// TIA Portal project "Project2" (V20)

(* hardware
DEVICE "S7-300/ET200M station_1"  S7-300 station
   slot 0: "Rail_0"  Rail  6ES7 390-1***0-0AA0
   slot 2: "PLC_1"  CPU 312  6ES7 312-1AE14-0AB0  V3.3
      slot 0: "MPI interface_1"  MPI
*)

// ===== PLC "PLC_1"  CPU 312 =====

ORGANIZATION_BLOCK "Main"   // OB1, LAD
TITLE = "Main Program Sweep (Cycle)"
{ S7_Optimized_Access := 'FALSE' }
VERSION : 0.1
   VAR_TEMP
      OB1_EV_CLASS : Byte;   // Bits 0-3 = 1 (Coming event), Bits 4-7 = 1 (Event class 1)
      OB1_SCAN_1 : Byte;   // 1 (Cold restart scan 1 of OB 1), 3 (Scan 2-n of OB 1)
      OB1_PRIORITY : Byte;   // Priority of OB Execution
      OB1_OB_NUMBR : Byte;   // 1 (Organization block 1, OB1)
      OB1_RESERVED_1 : Byte;   // Reserved for system
      OB1_RESERVED_2 : Byte;   // Reserved for system
      OB1_PREV_CYCLE : Int;   // Cycle time of previous OB1 scan (milliseconds)
      OB1_MIN_CYCLE : Int;   // Minimum cycle time of OB1 (milliseconds)
      OB1_MAX_CYCLE : Int;   // Maximum cycle time of OB1 (milliseconds)
      OB1_DATE_TIME : Date_And_Time;   // Date and time OB1 started
      S6 : Bool;
      S7 : Bool;
      S8 : Bool;
      "S1(sus stanga)" : Bool;
      "S2(sus Dreapta)" : Bool;
      "S3(jos stanga)" : Bool;
      "S4(jos Dreapta)" : Bool;
      "S5(soft reset)" : Bool;
      "S0(Hard reset)" : Bool;
      eroare : Bool;
      P1 : Bool;
      P2 : Bool;
      P3 : Bool;
      P4 : Bool;
      alarma : Bool;
   END_VAR
   VAR_TEMP   // added for the SCL form of the ladder/FBD networks
      _w1 : Bool;
      _w2 : Bool;
      _w3 : Bool;
      _w4 : Bool;
   END_VAR
BEGIN

REGION Network 1
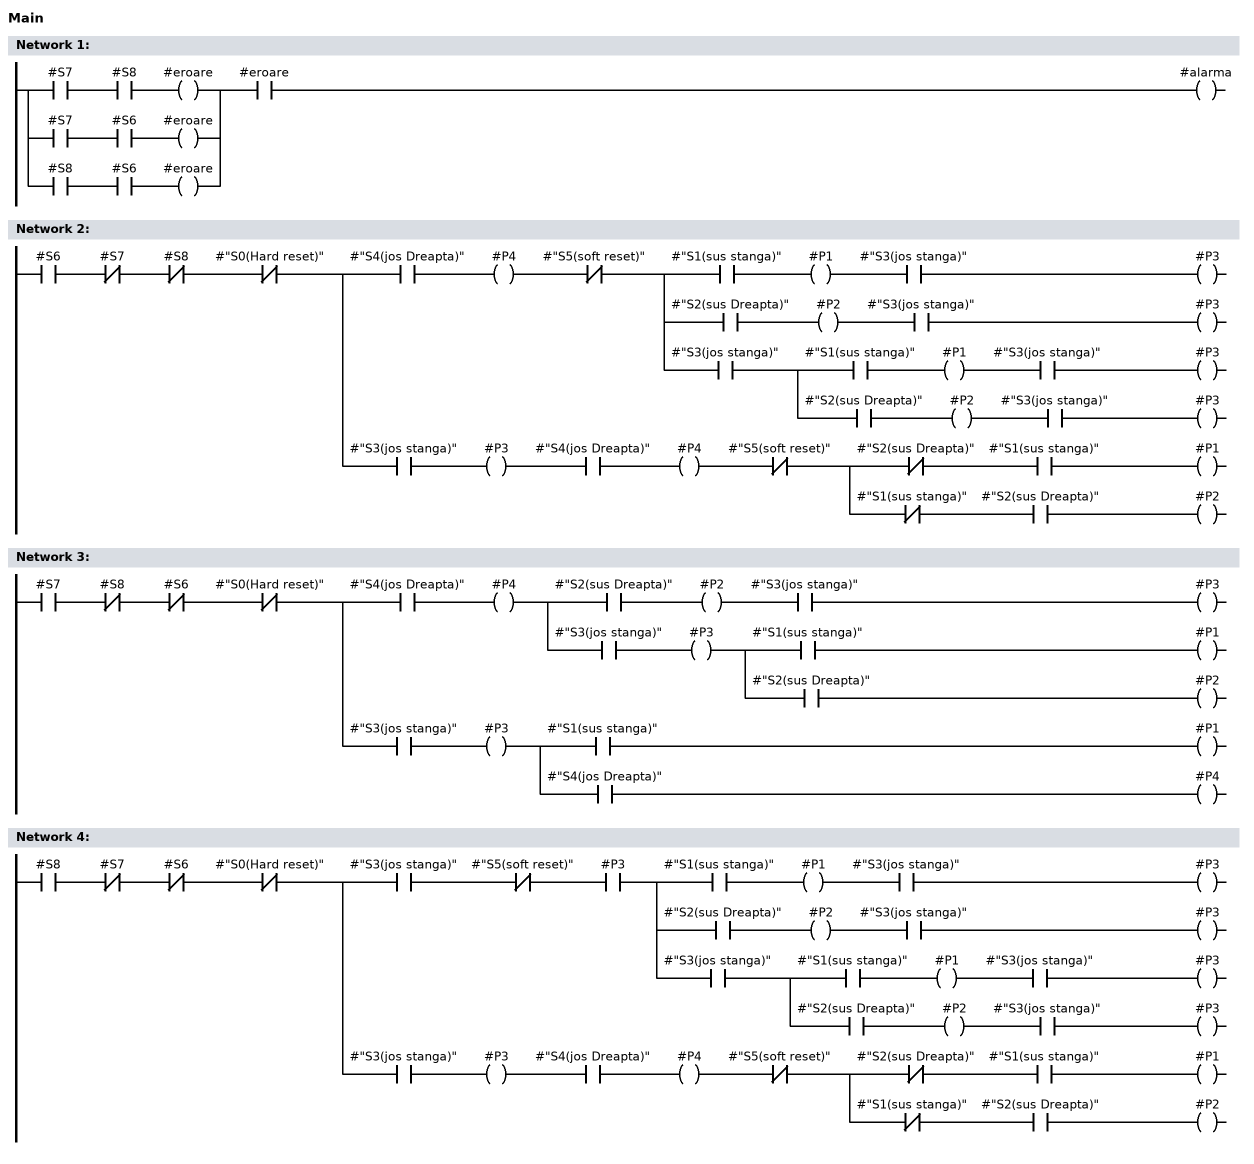
   RUNG wire#powerrail
      Contact( #S7 )
      Contact( #S8 )
      Coil( #eroare )
      wire#w1
      Contact( #eroare )
      Coil( #alarma )
   END_RUNG
   RUNG wire#powerrail
      Contact( #S7 )
      Contact( #S6 )
      Coil( #eroare )
   END_RUNG wire#w1
   RUNG wire#powerrail
      Contact( #S8 )
      Contact( #S6 )
      Coil( #eroare )
   END_RUNG wire#w1
   // the same network as SCL:
   #eroare := #S7 AND #S8;
   #_w1 := #eroare;
   #eroare := #S7 AND #S6;
   #_w2 := #eroare;
   #eroare := #S8 AND #S6;
   #alarma := (#_w1 OR #_w2 OR #eroare) AND #eroare;
END_REGION

REGION Network 2
   RUNG wire#powerrail
      Contact( #S6 )
      I_Contact( #S7 )
      I_Contact( #S8 )
      I_Contact( #"S0(Hard reset)" )
      wire#w1
      Contact( #"S4(jos Dreapta)" )
      Coil( #P4 )
      I_Contact( #"S5(soft reset)" )
      wire#w2
      Contact( #"S1(sus stanga)" )
      Coil( #P1 )
      Contact( #"S3(jos stanga)" )
      Coil( #P3 )
   END_RUNG
   RUNG wire#w2
      Contact( #"S2(sus Dreapta)" )
      Coil( #P2 )
      Contact( #"S3(jos stanga)" )
      Coil( #P3 )
   END_RUNG
   RUNG wire#w2
      Contact( #"S3(jos stanga)" )
      wire#w3
      Contact( #"S1(sus stanga)" )
      Coil( #P1 )
      Contact( #"S3(jos stanga)" )
      Coil( #P3 )
   END_RUNG
   RUNG wire#w3
      Contact( #"S2(sus Dreapta)" )
      Coil( #P2 )
      Contact( #"S3(jos stanga)" )
      Coil( #P3 )
   END_RUNG
   RUNG wire#w1
      Contact( #"S3(jos stanga)" )
      Coil( #P3 )
      Contact( #"S4(jos Dreapta)" )
      Coil( #P4 )
      I_Contact( #"S5(soft reset)" )
      wire#w4
      I_Contact( #"S2(sus Dreapta)" )
      Contact( #"S1(sus stanga)" )
      Coil( #P1 )
   END_RUNG
   RUNG wire#w4
      I_Contact( #"S1(sus stanga)" )
      Contact( #"S2(sus Dreapta)" )
      Coil( #P2 )
   END_RUNG
   // the same network as SCL:
   #_w1 := #S6 AND NOT #S7 AND NOT #S8 AND NOT #"S0(Hard reset)";
   #P4 := #_w1 AND #"S4(jos Dreapta)";
   #_w2 := #P4 AND NOT #"S5(soft reset)";
   #P1 := #_w2 AND #"S1(sus stanga)";
   #P3 := #P1 AND #"S3(jos stanga)";
   #P2 := #_w2 AND #"S2(sus Dreapta)";
   #P3 := #P2 AND #"S3(jos stanga)";
   #_w3 := #_w2 AND #"S3(jos stanga)";
   #P1 := #_w3 AND #"S1(sus stanga)";
   #P3 := #P1 AND #"S3(jos stanga)";
   #P2 := #_w3 AND #"S2(sus Dreapta)";
   #P3 := #P2 AND #"S3(jos stanga)";
   #P3 := #_w1 AND #"S3(jos stanga)";
   #P4 := #P3 AND #"S4(jos Dreapta)";
   #_w4 := #P4 AND NOT #"S5(soft reset)";
   #P1 := #_w4 AND NOT #"S2(sus Dreapta)" AND #"S1(sus stanga)";
   #P2 := #_w4 AND NOT #"S1(sus stanga)" AND #"S2(sus Dreapta)";
END_REGION

REGION Network 3
   RUNG wire#powerrail
      Contact( #S7 )
      I_Contact( #S8 )
      I_Contact( #S6 )
      I_Contact( #"S0(Hard reset)" )
      wire#w1
      Contact( #"S4(jos Dreapta)" )
      Coil( #P4 )
      wire#w2
      Contact( #"S2(sus Dreapta)" )
      Coil( #P2 )
      Contact( #"S3(jos stanga)" )
      Coil( #P3 )
   END_RUNG
   RUNG wire#w2
      Contact( #"S3(jos stanga)" )
      Coil( #P3 )
      wire#w3
      Contact( #"S1(sus stanga)" )
      Coil( #P1 )
   END_RUNG
   RUNG wire#w3
      Contact( #"S2(sus Dreapta)" )
      Coil( #P2 )
   END_RUNG
   RUNG wire#w1
      Contact( #"S3(jos stanga)" )
      Coil( #P3 )
      wire#w4
      Contact( #"S1(sus stanga)" )
      Coil( #P1 )
   END_RUNG
   RUNG wire#w4
      Contact( #"S4(jos Dreapta)" )
      Coil( #P4 )
   END_RUNG
   // the same network as SCL:
   #_w1 := #S7 AND NOT #S8 AND NOT #S6 AND NOT #"S0(Hard reset)";
   #P4 := #_w1 AND #"S4(jos Dreapta)";
   #P2 := #P4 AND #"S2(sus Dreapta)";
   #P3 := #P2 AND #"S3(jos stanga)";
   #P3 := #P4 AND #"S3(jos stanga)";
   #P1 := #P3 AND #"S1(sus stanga)";
   #P2 := #P3 AND #"S2(sus Dreapta)";
   #P3 := #_w1 AND #"S3(jos stanga)";
   #P1 := #P3 AND #"S1(sus stanga)";
   #P4 := #P3 AND #"S4(jos Dreapta)";
END_REGION

REGION Network 4
   RUNG wire#powerrail
      Contact( #S8 )
      I_Contact( #S7 )
      I_Contact( #S6 )
      I_Contact( #"S0(Hard reset)" )
      wire#w1
      Contact( #"S3(jos stanga)" )
      I_Contact( #"S5(soft reset)" )
      Contact( #P3 )
      wire#w2
      Contact( #"S1(sus stanga)" )
      Coil( #P1 )
      Contact( #"S3(jos stanga)" )
      Coil( #P3 )
   END_RUNG
   RUNG wire#w2
      Contact( #"S2(sus Dreapta)" )
      Coil( #P2 )
      Contact( #"S3(jos stanga)" )
      Coil( #P3 )
   END_RUNG
   RUNG wire#w2
      Contact( #"S3(jos stanga)" )
      wire#w3
      Contact( #"S1(sus stanga)" )
      Coil( #P1 )
      Contact( #"S3(jos stanga)" )
      Coil( #P3 )
   END_RUNG
   RUNG wire#w3
      Contact( #"S2(sus Dreapta)" )
      Coil( #P2 )
      Contact( #"S3(jos stanga)" )
      Coil( #P3 )
   END_RUNG
   RUNG wire#w1
      Contact( #"S3(jos stanga)" )
      Coil( #P3 )
      Contact( #"S4(jos Dreapta)" )
      Coil( #P4 )
      I_Contact( #"S5(soft reset)" )
      wire#w4
      I_Contact( #"S2(sus Dreapta)" )
      Contact( #"S1(sus stanga)" )
      Coil( #P1 )
   END_RUNG
   RUNG wire#w4
      I_Contact( #"S1(sus stanga)" )
      Contact( #"S2(sus Dreapta)" )
      Coil( #P2 )
   END_RUNG
   // the same network as SCL:
   #_w1 := #S8 AND NOT #S7 AND NOT #S6 AND NOT #"S0(Hard reset)";
   #_w2 := #_w1 AND #"S3(jos stanga)" AND NOT #"S5(soft reset)" AND #P3;
   #P1 := #_w2 AND #"S1(sus stanga)";
   #P3 := #P1 AND #"S3(jos stanga)";
   #P2 := #_w2 AND #"S2(sus Dreapta)";
   #P3 := #P2 AND #"S3(jos stanga)";
   #_w3 := #_w2 AND #"S3(jos stanga)";
   #P1 := #_w3 AND #"S1(sus stanga)";
   #P3 := #P1 AND #"S3(jos stanga)";
   #P2 := #_w3 AND #"S2(sus Dreapta)";
   #P3 := #P2 AND #"S3(jos stanga)";
   #P3 := #_w1 AND #"S3(jos stanga)";
   #P4 := #P3 AND #"S4(jos Dreapta)";
   #_w4 := #P4 AND NOT #"S5(soft reset)";
   #P1 := #_w4 AND NOT #"S2(sus Dreapta)" AND #"S1(sus stanga)";
   #P2 := #_w4 AND NOT #"S1(sus stanga)" AND #"S2(sus Dreapta)";
END_REGION
END_ORGANIZATION_BLOCK